// TwinCAT 3 PLC project PLC
// ProgramVersion: 3.1.4024.0
// libraries:
//   EfficientIO Communicator, * (EfficientIO)
//   Lynus Energy Basic, * (Lynus AG)
//   Tc2_Standard, * (Beckhoff Automation GmbH)
//   Tc2_System, * (Beckhoff Automation GmbH)
//   Tc2_Utilities, * (Beckhoff Automation GmbH)
//   Tc3_Module, * (Beckhoff Automation GmbH)
// project tree:
//   / FastTask.TcTTO, MiddleTask.TcTTO, SlowTask.TcTTO
//   POUs/ prgCom.TcPOU, prgMain.TcPOU, prgRWEffIO.TcPOU (not stored), prgVarEffIO.TcPOU (not stored)
// real-time tasks:
//   TASK FastTask: cycle T#5ms, priority 19, ADS port 350
//   TASK MiddleTask: cycle T#10ms, priority 20, ADS port 351
//   TASK SlowTask: cycle T#20ms, priority 21, ADS port 352
// I/O:
//   DEVICE Gerät 2 (CX-BK)
//     Box 1 (CX-BK)
// variable links:
//   PLC/PLC Instance <-> Device 2 (CX-BK)/Box 1 (CX-BK)
//     MiddleTask Inputs/prgMain.m_In1 <-> Term 3 (KL1408)/Channel 1/Eingang
//     MiddleTask Inputs/prgMain.m_In2 <-> Term 3 (KL1408)/Channel 2/Eingang
//     MiddleTask Outputs/prgMain.m_out1 <-> Term 2 (KL2408)/Channel 1/Ausgang

CONFIGURATION PLC
    RESOURCE PLC ON TwinCAT3
        TASK FastTask(INTERVAL := T#5ms, PRIORITY := 19);
        TASK MiddleTask(INTERVAL := T#10ms, PRIORITY := 20);
        TASK SlowTask(INTERVAL := T#20ms, PRIORITY := 21);
        PROGRAM prgRWEffIO WITH FastTask : prgRWEffIO;
        PROGRAM prgVarEffIO WITH FastTask : prgVarEffIO;
        PROGRAM prgMain WITH MiddleTask : prgMain;
        PROGRAM prgCom WITH SlowTask : prgCom;
    END_RESOURCE
END_CONFIGURATION

// ---- POUs/prgMain.TcPOU
PROGRAM prgMain
VAR
	m_Command_Himmelkron_RESET					: BOOL;							//{#lynus.ag#()}
	m_out1								AT%Q* 	: BOOL;
	r_tigt_Start_Reset: R_trig;
	tof_Reset: Tof;
	m_In1								AT%I* 	: BOOL;
	m_In2								AT%I* 	: BOOL;
	m_Input_Beacon_Himmelkorn					: BOOL;							//{#lynus.ag#()}
	m_Input_Siren_Himmelkorn					: BOOL;							//{#lynus.ag#()}
	m_LiveBit_5min_Himmelkorn								: BOOL;							//{#lynus.ag#()}
	ton_5Min: Ton;
END_VAR

r_tigt_Start_Reset( CLK := m_Command_Himmelkron_RESET);

tof_Reset(	IN:= r_tigt_Start_Reset.Q, 
			PT:= T#2S , 
			Q=> m_out1, 
			ET=> );

 
 m_Input_Beacon_Himmelkorn			:= 			m_In1;
 m_Input_Siren_Himmelkorn			:= 			m_In2;		// nicht ausgeführt
 
 
 ton_5Min(	In := NOT ton_5min.Q	,
	 		PT := T#5M);
			
IF ton_5min.Q AND m_LiveBit_5min_Himmelkorn THEN
	m_LiveBit_5min_Himmelkorn := FALSE;
ELSIF  ton_5min.Q AND NOT m_LiveBit_5min_Himmelkorn THEN
	m_LiveBit_5min_Himmelkorn := TRUE;
END_IF

END_PROGRAM

// ---- POUs/prgCom.TcPOU
PROGRAM prgCom
VAR
	fbCom		: FB_MqttCommunicator_V3;
	
	fb_Reboot		: NT_reboot;
	m_Reboot		: BOOL:=FALSE;
END_VAR

fbCom(
	bConnect:= TRUE, 
	strAuthKey					:=  'TSG88376368072' ,
	sUserName					:= '1d5b87ea-6e53-4c69-ac9d-4aea1f488196', 
	sUserPassword				:= '6a606077-744f-44bd-bbe1-ec67aa4d2e8c', 
	eSavePositionCertificate	:= eSavePositionOnPLC.ePostionHardDisk, 
	time_HeartBeat_sec 			:= T#30S,
	bConnected=> , 
	bError=> , 
	hrErrorCode=> , 
	eConnectionState=> , 
	eErrorMessage_Out=> );
	
	
fb_Reboot(	netid := '',
			delay := 2,
			start := m_Reboot);

END_PROGRAM
